Yaskawa INFORM job: FMTV_HOOD_BACK.JBI

/JOB
//NAME FMTV_HOOD_BACK
//POS
///NPOS 58,0,0,0,0,0
///TOOL 0
///POSTYPE PULSE
///PULSE
C00000=164501,-173796,-97080,-262022,121018,-52705
C00001=-144080,21368,-109469,-34247,107731,-96636
C00002=-144080,21368,-25913,-34247,107731,-96636
C00003=-151735,20733,-1708,-32098,94446,-95258
C00004=-151470,15625,-6510,-32114,94360,-95106
C00005=-155844,13002,-12158,-31278,95911,-92503
C00006=-157115,5561,-23309,-32456,90646,-90660
C00007=-163176,-2576,-31551,-32241,84903,-89048
C00008=-163154,-2752,-31647,-32249,84874,-89028
C00009=-165398,-7487,-37313,-32308,82489,-84765
C00010=-167563,-11045,-41642,-31867,81713,-80198
C00011=-169239,-14315,-44760,-31338,81158,-77084
C00012=-170419,-16629,-46728,-30962,80681,-75594
C00013=-170747,-17151,-47270,-30852,80602,-75232
C00014=-174623,-25647,-53446,-29858,78161,-74775
C00015=-179833,-35838,-59889,-28518,74653,-74317
C00016=-191818,-53869,-69609,-25181,66954,-74296
C00017=-191834,-53843,-69617,-25172,66965,-74306
C00018=-199545,-67879,-74424,-23207,60348,-59242
C00019=-202180,-77009,-74183,-23321,55179,-48829
C00020=-201091,-83275,-70005,-25454,50642,-43168
C00021=-199303,-80409,-69481,-25786,52279,-48304
C00022=-196387,-71271,-69255,-25551,57311,-65723
C00023=-203789,-77086,-71586,-23006,53501,-74177
C00024=-202758,-76384,-72487,-22316,53127,-86772
C00025=-230455,-90843,-75488,-34000,47529,-83224
C00026=-239939,-91694,-74758,-36255,46452,-83061
C00027=-240248,-87666,-77633,-34280,49207,-84700
C00028=-240533,-87133,-115999,-34103,49190,-84869
C00029=158635,-86033,-127751,-34103,49190,-84869
C00030=160360,-5327,-56177,-11633,96164,-95942
C00031=159095,15298,-20070,-7709,99070,-96206
C00032=158407,15976,-8598,-7556,93643,-96067
C00033=158616,11739,-12708,-7577,93546,-95981
C00034=162368,5091,-22692,-7836,88040,-99497
C00035=167232,-4901,-35316,-7408,80437,-104099
C00036=174428,-16224,-44817,-7658,70007,-105323
C00037=174431,-16201,-44809,-7659,70014,-105323
C00038=178397,-17996,-44873,-9375,69527,-108967
C00039=183551,-25850,-48120,-9154,64548,-119294
C00040=189084,-51428,-66404,9851,55635,-124593
C00041=200982,-61315,-70144,11376,61838,-130693
C00042=205878,-69891,-71070,9916,57799,-139439
C00043=204169,-75149,-69920,14496,54069,-141725
C00044=201289,-79082,-67895,19386,51309,-144657
C00045=203382,-78575,-70052,20275,51642,-134651
C00046=204553,-77826,-70973,19484,52333,-121403
C00047=204661,-77389,-72325,19206,53159,-112106
C00048=210023,-81931,-73222,29590,54330,-115703
C00049=215446,-84414,-72681,38309,56212,-118627
C00050=221260,-85232,-71204,45624,58447,-120825
C00051=226136,-84985,-69385,50800,60301,-122232
C00052=231482,-83751,-67060,55654,62307,-123338
C00053=232083,-80387,-69191,54410,63579,-121768
C00054=233872,-63521,-75041,50088,69749,-115793
C00055=232410,-167483,-107201,53740,64318,-120903
C00056=27737,-174553,-1120,-56108,-90364,-124885
C00057=-63952,-155163,126853,-105316,-81596,-126671
//INST
///DATE 2023/03/28 16:18
///ATTR SC,RW
///GROUP1 RB1
NOP
MOVJ C00000 VJ=65.00  //FROM RIGHT
MOVJ C00001 VJ=65.00
MOVJ C00002 VJ=65.00  //ABOVE RIGHT
MOVL C00003 V=65.0  //INLINE
MOVL C00004 V=15.0  //IN RIGHT SIDE
MOVL C00005 V=15.0
MOVL C00006 V=15.0
MOVL C00007 V=15.0
MOVC C00008 V=15.0
MOVC C00009 V=15.0
MOVC C00010 V=15.0
MOVC C00011 V=15.0
MOVC C00012 V=15.0
MOVC C00013 V=15.0
MOVL C00014 V=15.0
MOVL C00015 V=15.0
MOVL C00016 V=15.0
MOVC C00017 V=30.0
MOVC C00018 V=30.0
MOVC C00019 V=30.0
MOVL C00020 V=15.0
MOVL C00021 V=15.0
MOVL C00022 V=15.0
MOVL C00023 V=15.0
MOVL C00024 V=6.0
MOVL C00025 V=15.0
MOVL C00026 V=15.0  //END
MOVL C00027 V=65.0  //AWAY
MOVJ C00028 VJ=65.00
MOVJ C00029 VJ=65.00  //ROTATE
MOVL C00030 V=65.0
MOVL C00031 V=65.0
MOVL C00032 V=65.0  //INLINE
MOVL C00033 V=15.0  //INTO LEFT
MOVL C00034 V=15.0
MOVL C00035 V=15.0
MOVL C00036 V=15.0
MOVC C00037 V=15.0
MOVC C00038 V=15.0
MOVC C00039 V=15.0
MOVL C00040 V=15.0
MOVL C00041 V=15.0
MOVL C00042 V=15.0
MOVL C00043 V=15.0
MOVL C00044 V=15.0
MOVL C00045 V=10.0
MOVL C00046 V=3.0
MOVL C00047 V=8.0
MOVL C00048 V=15.0
MOVL C00049 V=15.0
MOVL C00050 V=15.0
MOVL C00051 V=15.0
MOVL C00052 V=15.0  //END
MOVL C00053 V=45.0  //OUT
MOVL C00054 V=65.0
MOVJ C00055 VJ=65.00
MOVJ C00056 VJ=65.00
MOVJ C00057 VJ=65.00  //HOME
END
